// TIA Portal V21 export
VAR_GLOBAL   // PLC tag table "K_Portata"
END_VAR
VAR_GLOBAL CONSTANT   // user constants
   K_Portata_PortataIngresso : Int := 1;   // Inputflow / Portataingresso
END_VAR
